(* IEC 61131-3 sources: CodesysTest/alpha/export/FBs/Components/Motors/Applied Motion/FB_AppliedMotionStepServoMBBase.pou, 1 file *)

(* ---- MoveDistance.m.st ---- *)
(*#-#-#-#-#-#-#-#-#-#---Declaration---#-#-#-#-#-#-#-#-#-#-#-#-#*)

//{warning 'add method implementation '}
METHOD MoveDistance
VAR_INPUT
    (*Distance to move in inches*)
    distance    : REAL;
    (*Acceleration in RPM/sec*)
    acceleration    : INT;
    (*Deceleration in RPM/sec*)
    deceleration    : INT;
    (*Velocity in .25RPM*)
    velocity    : INT;
END_VAR
(*#-#-#-#-#-#-#-#-#-#---Implementation---#-#-#-#-#-#-#-#-#-#-#-#-#*)
